TYPE ST_RecCmd ://过程纠偏
STRUCT
    bLock:				BOOL;	//纠偏外部锁定
	bAuto:				BOOL;	//纠偏自动
	bManual:           BOOL;  //纠偏手动
	bCentre:           BOOL;	//纠偏居中

END_STRUCT
END_TYPE

(* stored: Version 1.1.0.1, ProductVersion 3.1.4024.9
   DUT ST_RecCmd: Id {5cfa5300-e4b7-4578-8d0d-4e11e8af5f9b} *)
